FUNCTION_BLOCK COUNTER
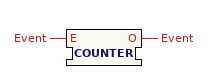
  EVENT_INPUT
    E;
  END_EVENT
  EVENT_OUTPUT
    O;
  END_EVENT
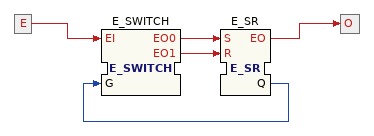
  FBS
    E_SWITCH : E_SWITCH;
    E_SR : E_SR;
  END_FBS
  EVENT_CONNECTIONS
    E_SWITCH.EO0 TO E_SR.S;
    E_SWITCH.EO1 TO E_SR.R;
    E_SR.EO TO O;
    E TO E_SWITCH.EI;
  END_CONNECTIONS
  DATA_CONNECTIONS
    E_SR.Q TO E_SWITCH.G;
  END_CONNECTIONS
END_FUNCTION_BLOCK
